(* LS Electric XG5000 project: 04_Practice2_1 *)
(* PLC LSPLC *)
(* module base 0 slot 0: 입력 모듈:XGI-D21A (DC 24V 입력, 8점 (전류소스/싱크입력)) *)
(* module base 0 slot 1: 출력 모듈:XGQ-RY1A (릴레이 출력, 8점 (2A용, 단독 COM.)) *)

PROGRAM NewProgram (* task: 스캔 프로그램 *)
VAR
    램프1 AT %QX0.1.0 : BOOL;
    램프2 AT %QX0.1.1 : BOOL;
    램프3 AT %QX0.1.2 : BOOL;
    램프4 AT %QX0.1.3 : BOOL;
    삼초 : TIME := T#3S;
    시작버튼 AT %IX0.0.0 : BOOL;
    타이머1 : TON;
    타이머2 : TON;
    타이머3 : TON;
    타이머4 : TON;
    타이머5 : TON;
END_VAR

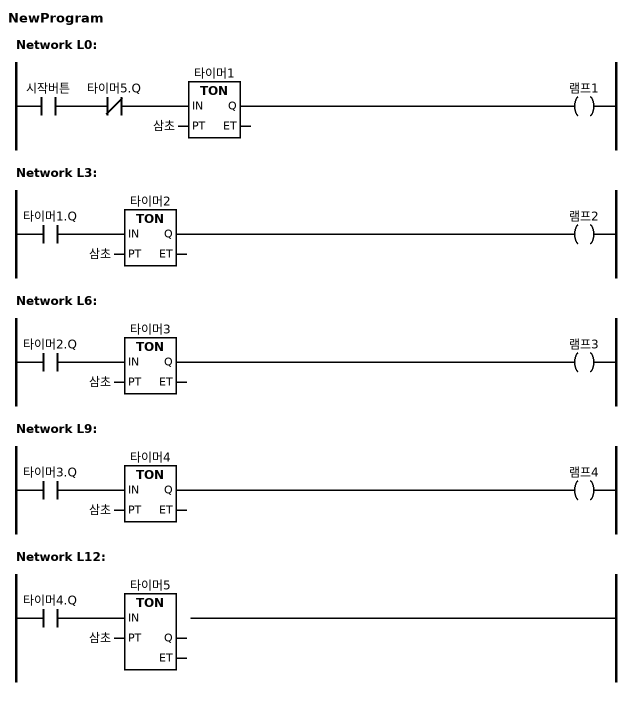
(* Rung L0 *)
타이머1(IN := 시작버튼 AND NOT 타이머5.Q, PT := 삼초);
램프1 := 타이머1.Q;
(* Rung L3 *)
타이머2(IN := 타이머1.Q, PT := 삼초);
램프2 := 타이머2.Q;
(* Rung L6 *)
타이머3(IN := 타이머2.Q, PT := 삼초);
램프3 := 타이머3.Q;
(* Rung L9 *)
타이머4(IN := 타이머3.Q, PT := 삼초);
램프4 := 타이머4.Q;
(* Rung L12 *)
타이머5(IN := 타이머4.Q, PT := 삼초);
END_PROGRAM